(*
Used by Start() to return an error indication. Cannot use the host object without interfering with the current execution.
*)
{attribute 'reflection'}
FUNCTION_BLOCK T_ExecutionInError IMPLEMENTS I_ExecutionResult
VAR
    _State    : T_ExecutionState;
    _Done     : BOOL;
    _Error    : BOOL;
    _Aborted  : BOOL;
    _ErrorMsg : T_MaxString;

    {attribute 'instance-path'}
    {attribute 'no_init'}
    Name     : T_MaxString; // Automatically initialised with the full name of the instance
    Project  : T_MaxString;
    Solution : T_MaxString;

    _Notification_OnError : I_Notification;
    _Notification_OnAbort : I_Notification;
    _Logger               : I_Logger;
END_VAR

METHOD Abort
VAR_INPUT
END_VAR
// Not implemented
END_METHOD

PROPERTY Aborted : BOOL
GET
Aborted := _Aborted;
END_GET
END_PROPERTY

PROPERTY Aborting : BOOL
GET
Aborting := _State = T_ExecutionState.Aborting;
END_GET
END_PROPERTY

PROPERTY Busy : BOOL
GET
Busy := _State = T_ExecutionState.Busy;
END_GET
END_PROPERTY

PROPERTY Done : BOOL
GET
Done := _Done;
END_GET
END_PROPERTY

PROPERTY Error : BOOL
GET
Error := _Error;
END_GET
END_PROPERTY

PROPERTY ErrorMsg : T_MaxString
GET
ErrorMsg := _ErrorMsg;
END_GET
END_PROPERTY

// Individual T_Execution events are assigned here to the global events 
// so by default, all errors/aborts raise these global events
// This can be overidden for individual instances or T_Execution 
// by setting the Event properties to zero (or another event)
METHOD FB_init : BOOL
VAR_INPUT
    bInitRetains : BOOL; // if TRUE, the retain variables are initialized (warm start / cold start)
    bInCopyCode  : BOOL; // if TRUE, the instance afterwards gets moved into the copy code (online change)
END_VAR
VAR
    StringSplitter : T_StringSplitter;
END_VAR
_Notification_OnAbort := GlobalNotifications.Notification_ExecutionAborted;
_Notification_OnError := GlobalNotifications.Notification_ExecutionFailed;
_Logger               := GlobalNotifications.Logger;

StringSplitter.Init(Str    := Name,
                    Delim1 := '.',
                    Delim2 := '');

Solution := StringSplitter.GetNext();
Project  := StringSplitter.GetNext();
Name     := StringSplitter.GetRemainder();
END_METHOD

PROPERTY Ready : BOOL
GET
Ready := _State = T_ExecutionState.Ready;
END_GET
END_PROPERTY

METHOD SetError
VAR_INPUT
    ErrorMsg : T_MaxString;
END_VAR
VAR
    pSTRING : POINTER TO STRING;
    arg     : T_Arg;
END_VAR
IF NOT _Error THEN // ignore subsequent errors in an execution sequence
    _Error    := TRUE;
    _Aborted  := FALSE;
    _Done     := FALSE;
    _ErrorMsg := ErrorMsg;
    _State    := T_ExecutionState.Ready;

    IF _Notification_OnError <> 0 THEN
        _Notification_OnError.Args
            .Clear()
            .Add_STRING(_ErrorMsg)
            .Add_STRING(Name);

        _Notification_OnError.Raise();
    END_IF

    IF _Logger <> 0 THEN
        _Logger.LogError(Source := Name, Message := _ErrorMsg);
    END_IF

END_IF
END_METHOD

PROPERTY Starting : BOOL
GET
Starting := _State = T_ExecutionState.Starting;
END_GET
END_PROPERTY

END_FUNCTION_BLOCK

(* stored: Version 1.1.0.1, ProductVersion 3.1.4024.12
   POU T_ExecutionInError: Id {1b10dd92-5b6d-46bf-969d-2d1571e3af65}, SpecialFunc None
   Folder Methods: Id {85cb006e-7eaa-4f5f-bb05-e9c5af191c83}
   Folder Properties: Id {df36a550-4c05-4c4b-a5cb-af57421e91d0}
   Method Abort: Id {6f99ecc8-8720-46c8-8a4f-6b24c96ac05f}
   Property Aborted: Id {02cb6069-7582-4125-b1f8-d0d2aa43deb5}
   Get Get: Id {e8225a2c-dcf4-43c4-a793-f827674aa675}
   Property Aborting: Id {4078d57f-38d4-4706-9acb-ca79bed5f1ab}
   Get Get: Id {0bf9c612-f46e-4474-a73d-64fd31fee069}
   Property Busy: Id {0f619bd1-4466-427b-92e4-2804ff599614}
   Get Get: Id {43116eaa-18c1-4783-95c7-e4a2702a609d}
   Property Done: Id {de4f204a-7ff6-4704-9f2d-7cc6100cef5f}
   Get Get: Id {7825cecc-4ac9-4bb1-bc86-0db5b8ec8816}
   Property Error: Id {8a7c8a41-5022-4dc9-8de8-1074dbe83b1b}
   Get Get: Id {23eb850c-a4e4-40ab-b230-dc9f361029ca}
   Property ErrorMsg: Id {0ca0f1ab-980d-4b87-bed5-02001ca05df9}
   Get Get: Id {8d4d1d29-4c27-4933-a0a2-0831b5136711}
   Method FB_init: Id {ef66a107-056e-4ecb-8b6e-7ea45b73f6f7}
   Property Ready: Id {37328bdd-550f-4c87-8fd6-17d906073889}
   Get Get: Id {2a0e3a7b-dd92-433b-a09a-6273f1f9cedc}
   Method SetError: Id {9230d86b-408b-456c-8f86-609961b0a0b9}
   Property Starting: Id {289bfee9-f1c8-413e-9f32-578bce6d3b9a}
   Get Get: Id {680679f0-d3b8-45a0-a116-54fb5a269ae0} *)
